TYPE OperatorInfo EXTENDS TcoCore.TcoStruct :
STRUCT
	UserName : STRING(255);
END_STRUCT
END_TYPE

(* stored: Version 1.1.0.1
   DUT OperatorInfo: Id {e8f1a1f6-3458-4107-ab96-c9cf5a6b2384} *)
